FUNCTION_BLOCK PneumaticInsertion// EXTENDS Insertion
VAR_INPUT
	enable : BOOL;
END_VAR
VAR_OUTPUT
	slider : ClearLinkEIP;
	screw : AirPiston;
	
	contact : BOOL;
	
	home : BOOL;
	ready : BOOL;
	busy : BOOL;
	error : BOOL;
	
	homeSet : BOOL;
END_VAR

slider(
	bEnable:= enable, 
	home=> , 
	outerLimit=> , 
	innerLimit=> , 
	contact=> contact, 
	homeSet=> );
	
screw(
	bEnable:= enable,
	valveIn=> , 
	valveOut=> , 
	contact=> , 
	home=> , 
	innerLimit=> , 
	ready=> , 
	busy=> , 
	error=> , 
	homeSet=> );
	
home := screw.home AND slider.home;
busy := slider.busy OR screw.busy;
error := slider.error OR screw.error;

homeSet := slider.homeSet AND screw.homeSet;

METHOD homingSequence : BOOL
IF NOT screw.homeSet THEN
	screw.homingSequence();
END_IF

homingSequence := slider.homeSet (*AND screw.homeSet*);
END_METHOD

METHOD press : BOOL
VAR_INPUT
	//direction : BOOL; //direction (F = inwards, T = outwards)
	//distance : DINT;
END_VAR
press := screw.slideIn();
END_METHOD

METHOD release : BOOL
VAR_INPUT
END_VAR
release := screw.slideOut();
END_METHOD

METHOD slideAbsolute : BOOL
VAR_INPUT
	targetPos : REAL;
END_VAR
slideAbsolute := slider.moveAbsolute(newTarget:= targetPos);
END_METHOD

METHOD slideContinuous : BOOL
VAR_INPUT
	direction : MC_Direction;
END_VAR
slideContinuous := slider.moveContinuous(direction := direction);
END_METHOD

METHOD stop : BOOL
VAR_INPUT
END_VAR
slider.stop();
screw.stop();
END_METHOD

END_FUNCTION_BLOCK

(* stored: Version 1.1.0.1, ProductVersion 3.1.4024.11
   POU PneumaticInsertion: Id {b81c5df3-3bac-4f9d-9b77-7bbeccd1dc76}, SpecialFunc None
   Method homingSequence: Id {d7cd42ba-bf91-49d9-b290-abbbea3d3ad6}
   Method press: Id {b1e47417-f59e-4f47-a453-5b14f0c0ab9e}
   Method release: Id {6735797f-0df0-46da-8234-935ba24cde58}
   Method slideAbsolute: Id {89be0205-36be-4635-bf1d-734fb40c3796}
   Method slideContinuous: Id {b7ff75db-864c-438f-bfb9-1fb8fcf5dcaf}
   Method stop: Id {50e4fe0e-754b-400a-bf2a-178124b95404} *)
